TYPE ST_BaseHMIConnectorEvents_Filter :
STRUCT
	bActive						: BOOL;
	bNotActive					: BOOL;
	
	bIDItem						: BOOL;
	uiIDItem					: UINT;
	
	bIDEvent					: BOOL;
	uiIDEvent					: UINT;
	
	arrSelectedEventCategory	: ARRAY [0..GVL_BaseConstans.NUMBER_OF_EVENT_CATEGORIES] OF BOOL;
	
END_STRUCT
END_TYPE

(* stored: Version 1.1.0.1
   DUT ST_BaseHMIConnectorEvents_Filter: Id {0a75babb-bdad-091c-1ce3-1452b30582ad} *)
